Staubli VAL3: clkValve12.pgx

program clkValve12()
begin
  call toggleValve(12)
end
